(* IEC 61131-3 sources: vscode-twincat-st/src/sample/Base, 18 files *)

(* ---- Comments.st ---- *)
// This is my struct.
TYPE ST_Comments :
STRUCT
    // a
    a: BOOL := FALSE; // My Comment

    // unused

    (* b
    b *)
    b: BOOL;

	c: BOOL; (*c
    c*)
END_STRUCT
END_TYPE

(* ---- GlobalVariableLists.st ---- *)
VAR_GLOBAL MyGVL
	A: INT;

	B: INT;
END_VAR

(* ---- Interfaces.st ---- *)
INTERFACE MyInterface

    PROPERTY MyValue : INT
        GET
            //
        END_GET
        SET
            //
        END_SET
    END_PROPERTY

    METHOD MyMethod : BOOL
        //
    END_METHOD
END_INTERFACE

(* ---- Functions.st ---- *)
FUNCTION MyFunction

    VAR_INPUT
        var_a: BOOL;
    END_VAR

    var_a := TRUE;
END_FUNCTION

(* ---- AccessModifiers.st ---- *)
PROGRAM INTERNAL AccessModifier
    //
END_PROGRAM

INTERFACE INTERNAL I_AccessModifier
    //
END_INTERFACE

FUNCTION_BLOCK INTERNAL FB_AccessModifier

    METHOD PRIVATE M_AccessModifier : INT
        //
    END_METHOD

    PROPERTY INTERNAL P_AccessModifier : INT
        GET PRIVATE
            //
        END_GET
        SET PRIVATE
            //
        END_SET
    END_PROPERTY
END_FUNCTION_BLOCK

FUNCTION INTERNAL F_AccessModifier : BOOL
    //
END_FUNCTION

TYPE INTERNAL A_AccessModifier : INT;
    //
END_TYPE

TYPE INTERNAL E_AccessModifier :
(
    dummy
);
END_TYPE

TYPE INTERNAL ST_AccessModifier :
STRUCT
    //
END_STRUCT
END_TYPE

TYPE INTERNAL U_AccessModifier :
UNION
    //
END_UNION
END_TYPE

VAR_GLOBAL INTERNAL GVL_AccessModifier
    //
END_VAR

(* ---- Arrays.st ---- *)
VAR_GLOBAL CONSTANT GVL_Array
    UPPER_LIMIT : INT := 1;
END_VAR

FUNCTION_BLOCK FB_Array
    VAR
        array: ARRAY [0+1..GVL_Array.UPPER_LIMIT] OF INT;
    END_VAR
END_FUNCTION_BLOCK

(* ---- Assignments.st ---- *)
FUNCTION_BLOCK Assignments

    VAR
        a: BOOL;
    END_VAR

    a := FALSE;
END_FUNCTION_BLOCK

(* ---- Constants.st ---- *)
VAR_GLOBAL CONSTANT GVL_Constants
	A: INT;
END_VAR

FUNCTION_BLOCK FB_Constants

    VAR
        _a: INT;
    END_VAR

    VAR_INPUT CONSTANT
        A: INT;
    END_VAR

    _a := A;
    _a := GVL_Constants.A;
END_FUNCTION_BLOCK

(* ---- FunctionBlocks.st ---- *)
FUNCTION_BLOCK MyFunctionBlock

    VAR_INPUT
        var_a: BOOL := FALSE;
    END_VAR

    PROPERTY MyValue : INT
        GET
            //
        END_GET
        SET
            //
        END_SET
    END_PROPERTY

    METHOD MyMethod : BOOL
        //
    END_METHOD

    var_a := TRUE;
END_FUNCTION_BLOCK

(* ---- ImplicitConversions.st ---- *)
// https://infosys.beckhoff.com/english.php?content=../content/1033/tf5100_tc3_nc_i/4188351883.html&id=

TYPE E_ImplicitConversions_Default :
(
    A
);
END_TYPE

TYPE E_ImplicitConversions_USINT :
(
    A
) SINT;
END_TYPE

TYPE InnerAlias : E_ImplicitConversions_USINT;
END_TYPE

TYPE OuterAlias : InnerAlias;
END_TYPE

FUNCTION_BLOCK ImplicitConversions

    VAR
        _uint:          UINT;
        _word:          WORD;
        _enum_default:  E_ImplicitConversions_Default   := 1;
        _enum_usint:    E_ImplicitConversions_USINT     := 1;
        _alias:         OuterAlias                      := 1;
        _assign_from_x: INT                             := E_ImplicitConversions_Default.A;
    END_VAR

    _uint           := _word;
    _enum_default   := 1;
    _enum_usint     := 1;
    _alias          := 1;
    _assign_from_x  := E_ImplicitConversions_Default.A;
    _assign_from_x  := _enum_default;
    _assign_from_x  := _alias;
END_FUNCTION_BLOCK

(* ---- Literals.st ---- *)
FUNCTION_BLOCK Literals

    VAR

        // Logical Types
        bool_0:                 BOOL            := 0;
        bool_false:             BOOL            := FALSE;
        bool_1:                 BOOL            := 1;
        bool_true:              BOOL            := TRUE;
        bool_typed:             BOOL            := BOOL#1;

        bit_0:                  BIT             := 0;
        bit_false:              BIT             := FALSE;
        bit_1:                  BIT             := 1;
        bit_true:               BIT             := TRUE;
        bit_typed:              BIT             := BIT#1;

        // Bitstring Types
        _word_1:                WORD            := 1;
        _word_2:                WORD            := 16#FFFF;

        // Unsigned Integer Types
        uint_positive:          UINT            := 010;
        uint_typed:             UINT            := UINT#1;
        usint_underscore:       UINT            := USINT#2__5_5;

        int_positive:           INT             := 10;
        int_negative:           INT             := -10;
        int_typed:              INT             := INT#-1;

        // HEX
        int_hex:                INT             := 16#0A;
        int_hex_typed:          INT             := INT#16#FF;

        // DEC
        int_dec:                INT             := 10#10;
        int_hdec_typed:         INT             := INT#10#255;

        // OCTAL
        int_octal:              INT             := 8#12;
        int_octal_typed:        INT             := INT#8#77;

        // BINARY
        int_binary:             INT             := 2#1010;
        int_binary_typed:       INT             := INT#2#11111111;

        // Floating Point Types
        real_int:               REAL            := 199;
        real_positive:          REAL            := REAL#1.99;
        real_negative:          REAL            := -1.99;
        real_scientific:        REAL            := 1e-99;
        real_underscore:        REAL            := 1__00e-9__9;

        // String Types
        string_narrow:          STRING          := 'A';
        string_narrow2:         STRING(1)       := 'A';
        string_wide:            WSTRING         := "Ā";
        string_wide2:           WSTRING(1)      := "Ā";

        // Time-Related Types

        // => TIME
        time_max:               TIME            := TIME#49D17H2M47S295MS;
        time_firstover:         TIME            := TIME#90H10MS;
        time_alt:               TIME            := T#05H10MS;

        // => LTIME
        l_time_max:             LTIME           := LTIME#213503D23H34M33S709MS551US615NS;
        l_time_firstover:       LTIME           := LTIME#90H10MS;
        l_time_alt:             LTIME           := LTIME#05H10MS;

        // => DATE: Nothing is optional
        date_min:               DATE            := DATE#1970-01-01;
        date_max:               DATE            := DATE#2106-02-07;
        date_min_alt:           DATE            := D#1970-01-001;

        // => LDATE: Nothing is optional
        l_date_min:             LDATE           := LDATE#1970-01-01;
        l_date_max:             LDATE           := LDATE#2554-7-21;
        l_date_min_alt:         LDATE           := LD#1970-1-001;

        // => TIME_OF_DAY: Milliseconds and seconds are optional
        time_of_day_min:        TIME_OF_DAY     := TIME_OF_DAY#0:0:0;
        time_of_day_max:        TIME_OF_DAY     := TIME_OF_DAY#23:59:59.999;
        time_of_day_alt:        TOD             := TOD#0:0;

        // => LTIME_OF_DAY: Milliseconds and seconds are optional
        l_time_of_day_min:      LTIME_OF_DAY    := LTIME_OF_DAY#0:0:0;
        l_time_of_day_max:      LTIME_OF_DAY    := LTIME_OF_DAY#23:59:59.999999999;
        l_time_of_day_alt:      LTOD            := LTOD#0:0;

        // => DATE_AND_TIME: Seconds are optional
        date_and_time_min:      DATE_AND_TIME   := DATE_AND_TIME#1970-1-1-0:0:0;
        date_and_time_max:      DATE_AND_TIME   := DATE_AND_TIME#2106-02-07-06:28:15;
        date_and_time_alt:      DT              := DT#1970-1-001-0:0;

        // => LDATE_AND_TIME: Milliseconds and seconds are optional
        l_date_and_time_min:    LDATE_AND_TIME  := LDATE_AND_TIME#1970-01-01-00:00:00;
        l_date_and_time_max:    LDATE_AND_TIME  := LDATE_AND_TIME#2554-7-21-23:34:33.709551615;
        l_date_and_time_alt:    LDT             := LDT#1970-1-001-0:0;
    END_VAR
END_FUNCTION_BLOCK

(* ---- MemberQualifiers.st ---- *)
TYPE E_MemberQualifier :
(
    Variable
);
END_TYPE

FUNCTION F_MemberQualifier : INT
    //
END_FUNCTION

VAR_GLOBAL GVL_MemberQualifier
    A: MemberQualifier_A;

    Variable: INT;
END_VAR

FUNCTION_BLOCK MemberQualifier_A

    VAR_INPUT
        Variable: INT;
    END_VAR

    METHOD MyMethod : INT
        //
    END_METHOD
END_FUNCTION_BLOCK

FUNCTION_BLOCK MemberQualifier_B

    VAR_OUTPUT
        A: MemberQualifier_A;

        Variable: INT;
    END_VAR

    METHOD MyMethod
        //
    END_METHOD
END_FUNCTION_BLOCK

FUNCTION_BLOCK MemberQualifier

    VAR
        _variable: INT;
        _b1: MemberQualifier_B;
    END_VAR

    METHOD MyMethod

        VAR
            variable: INT;
            _b2: MemberQualifier_B;
        END_VAR

        // Assignments + Expressions
        variable := variable;

        variable := _variable;
        variable := THIS^._variable;

        variable := E_MemberQualifier.Variable;

        // Call statements
        _b1();
        _b2();
        MyMethod();
        THIS^.MyMethod();

        F_MemberQualifier();
    END_METHOD

    METHOD MyMethod2 : INT
        //
    END_METHOD

    // Assignments + Expressions (variable usage and method/function usage)
    _variable := _variable;
    _variable := THIS^._variable;

    _variable := THIS^._b1.Variable;
    _variable := _b1.Variable;
    _variable := _b1.A.Variable;

    _variable := GVL_MemberQualifier.Variable;
    _variable := GVL_MemberQualifier.A.Variable;
    _variable := E_MemberQualifier.Variable;

    _variable := _b1.A.MyMethod();
    _variable := F_MemberQualifier();

    _b1.A.Variable := 1;

    // Call statements
    _b1();
    MyMethod();
    MyMethod2();
    THIS^.MyMethod();

    THIS^._b1.MyMethod();
    _b1.MyMethod();
    _b1.A.MyMethod();

    GVL_MemberQualifier.A.MyMethod();
    F_MemberQualifier();
END_FUNCTION_BLOCK

(* ---- Operators.st ---- *)
FUNCTION_BLOCK FB_Operators

    VAR
        // Unary
        _minus: BYTE := -BYTE#1;
        _plus:  BYTE := +BYTE#1;
        _not:   BYTE := NOT BYTE#1;

        // Binary
        _uint1: UINT := UINT#10 + 3;
        _uint2: UINT := UINT#10 - 3;
        _uint3: UINT := UINT#10 / 3;
        _uint4: UINT := UINT#10 * 3;

        // _uint5: UINT := UINT#10 / 0;
    END_VAR
END_FUNCTION_BLOCK

(* ---- References.st ---- *)
FUNCTION_BLOCK Referenced

    METHOD MyMethod

        VAR_INPUT
            a: REFERENCE TO INT;
        END_VAR
    END_METHOD
END_FUNCTION_BLOCK

FUNCTION_BLOCK References

    VAR
        original: Referenced;
        ref: REFERENCE TO Referenced REF= original;
        ptr: POINTER TO Referenced := ADR(original);

        myInt: INT;
        crazy1: POINTER TO ARRAY [0..1] OF POINTER TO ARRAY [0..1] OF ARRAY [0..1] OF POINTER TO POINTER TO INT;
        crazy2: POINTER TO ARRAY [0..1] OF POINTER TO ARRAY [0..1] OF ARRAY [0..1] OF POINTER TO POINTER TO Referenced;
    END_VAR

    // Referencing
    ref REF= original;
    ptr := ADR(original);

    original.MyMethod(a := myInt);

    // Dereferencing
    original    := ref;
    original    := ptr^;
    myInt       := crazy1^[0]^[0][0]^^;
    original    := crazy2^[0]^[0][0]^^;
END_FUNCTION_BLOCK

(* ---- Statements.st ---- *)
FUNCTION_BLOCK FB_Assignment

    VAR_INPUT
        a: INT;

        b: INT;
    END_VAR

    PROPERTY P_A : INT
        SET
            //
        END_SET
    END_PROPERTY
END_FUNCTION_BLOCK

FUNCTION_BLOCK Statements

    VAR
        assignment: FB_Assignment;
    END_VAR

    // Assignment
    assignment.a := b;
    assignment.P_A := b;
END_FUNCTION_BLOCK

(* ---- Subrange.st ---- *)
FUNCTION_BLOCK Subrange

    VAR
        _a: BYTE(0..0);
        _b: UINT(1..0);
        _c: INT(-4095..4095);
    END_VAR
END_FUNCTION_BLOCK

(* ---- TypeUsages.st ---- *)
FUNCTION_BLOCK FB_TypeUsage
    //
END_FUNCTION_BLOCK

TYPE ST_TypeUsage :
STRUCT
    A: BOOL;
END_STRUCT
END_TYPE

TYPE E_TypeUsage :
(
    A
);
END_TYPE

INTERFACE I_TypeUsage
    //
END_INTERFACE

FUNCTION_BLOCK TypeUsage

    VAR
        _functionBlock: FB_TypeUsage;
        _struct: ST_TypeUsage;
        _enum: E_TypeUsage;
        _interface: I_TypeUsage;
        _bool: BOOL;
    END_VAR
END_FUNCTION_BLOCK

(* ---- Programs.st ---- *)
PROGRAM Program
    //
END_PROGRAM
